// TIA Portal V20 export
DATA_BLOCK "CallEquipment_DB"   // DB18
{ DB_Accessible_From_OPC_UA := 'FALSE' }
// stored: AssignedProDiagFB Unit1.Em2.ProDiag, DBAccessibleFromOPCUA false, DBAccessibleFromWebserver false, InstanceOfName Unit1.Em2.CallEquipment, InstanceOfType FB, Namespace Unit1.Em2
"Unit1.Em2.CallEquipment"
   // VAR_INPUT
   //    ZoneOperationEnable { ExternalWritable := 'False'} : "LWONIK_typeSafetyZoneManualOperation";
   // END_VAR
   // VAR_IN_OUT
   //    unitStatus : "LAF_typeUnitStatus";
   //    emFeedback : "LUC_typeEmFeedback";
   //    unitAlarmDB : "LAF_typeAlarms";
   // END_VAR
   // VAR
   //    InstSequenceJROutPnPLeft { ExternalWritable := 'False'} : "Unit1.Em2.Sequence_1_JROutPnPLeft";
   //    InstSequenceJROutPnPRight { ExternalWritable := 'False'} : "Unit1.Em2.Sequence_2_JROutPnPRight";
   //    instJROutPnPLeftHomeJob1 { ExternalWritable := 'False'} : "LAF_SelectJob";
   //    instJROutPnPLeftStack1LoadJob2 { ExternalWritable := 'False'} : "LAF_SelectJob";
   //    instJROutPnPLeftStack2LoadJob3 { ExternalWritable := 'False'} : "LAF_SelectJob";
   //    instJROutPnPLeftUnloadJob4 { ExternalWritable := 'False'} : "LAF_SelectJob";
   //    instJROutPnPRightHomeJob1 { ExternalWritable := 'False'} : "LAF_SelectJob";
   //    instJROutPnPRightLoadJob2 { ExternalWritable := 'False'} : "LAF_SelectJob";
   //    instJROutPnPRightUnloadJob3 { ExternalWritable := 'False'} : "LAF_SelectJob";
   //    instCmJROutPnPLeftSafetyPin { ExternalWritable := 'False'} : "LBC_DigitalSignalCn";
   //    instCmJROutPnPLeftJRDetect { ExternalWritable := 'False'} : "LBC_DigitalSignalCn";
   //    instCmJROutPnPRightSafetyPin { ExternalWritable := 'False'} : "LBC_DigitalSignalCn";
   //    instCmJROutPnPRightJRDetect { ExternalWritable := 'False'} : "LBC_DigitalSignalCn";
   //    instCmJROutPnPLeftAxisX { ExternalWritable := 'False'} : "LBC_Axis64Pos_TecPlcCn";
   //    instCmJROutPnPLeftAxisZ { ExternalWritable := 'False'} : "LBC_Axis64Pos_TecPlcCn";
   //    instCmJROutPnPRightAxisX { ExternalWritable := 'False'} : "LBC_Axis64Pos_TecPlcCn";
   //    instCmJROutPnPRightAxisZ { ExternalWritable := 'False'} : "LBC_Axis64Pos_TecPlcCn";
   //    instCmJROutPnPLeftClampOpenClose { ExternalWritable := 'False'} : "LBC_TwoWayActuatorCn";
   //    instCmJROutPnPRightClampOpenClose { ExternalWritable := 'False'} : "LBC_TwoWayActuatorCn";
   //    instPowerMeter { ExternalWritable := 'False'} : "LER_PowerMeter_7KM";
   //    instInterlockJROutPnPLeftAxisX { ExternalWritable := 'False'} : "LER_Axis64Pos_InterlockSummary";
   //    instInterlockJROutPnPLeftAxisZ { ExternalWritable := 'False'} : "LER_Axis64Pos_InterlockSummary";
   //    instInterlockJROutPnPRightAxisX { ExternalWritable := 'False'} : "LER_Axis64Pos_InterlockSummary";
   //    instInterlockJROutPnPRightAxisZ { ExternalWritable := 'False'} : "LER_Axis64Pos_InterlockSummary";
   //    instLDrv701ControlJROutPnPLeftAxisZ { ExternalWritable := 'False'} : "LDrvSafe_SinaTlg701Control";
   //    instLDrv701StatusJROutPnPLeftAxisZ { ExternalWritable := 'False'} : "LDrvSafe_SinaTlg701Status";
   //    instLDrv701ControlJROutPnPRightAxisZ { ExternalWritable := 'False'} : "LDrvSafe_SinaTlg701Control";
   //    instLDrv701StatusJROutPnPRightAxisZ { ExternalWritable := 'False'} : "LDrvSafe_SinaTlg701Status";
   //    instEmOverviewHomeCondtion { ExternalWritable := 'False'} : "Unit1.Em2.LER_EmOverviewHomeCondtion";
   //    instManageAlarms { ExternalWritable := 'False'} : "LAF_ManageAlarms";
   //    instEventsPFE { ExternalWritable := 'False'} : "Unit1.Em2.EventsPFE";
   //    statUnitStatus { ExternalWritable := 'False'} : "LAF_typeUnitStatus";
   //    statSlmStatus { ExternalWritable := 'False'} : Struct
   //       running : Bool;
   //       powerOff : Bool;
   //    END_STRUCT;
   //    statAllBrakeTest { ExternalWritable := 'False'} : "LER_typeBrakeTestUnitCommands";
   //    statTonTime { ExternalWritable := 'False'} : Array[0..999] of TON_TIME;
   //    statTofTime { ExternalWritable := 'False'} : Array[0..99] of TOF_TIME;
   //    statReal { ExternalWritable := 'False'} : Array[0..19] of Real;
   //    statDWord { ExternalWritable := 'False'} : Array[0..9] of DWord;
   //    Static_1 { ExternalWritable := 'False'} : DWord;
   //    statDInt { ExternalWritable := 'False'} : Array[0..9] of DInt;
   //    statPulse { ExternalWritable := 'False'} : Array[0..999] of Bool;
   //    statFlipFlop { ExternalWritable := 'False'} : Array[0..99] of Bool;
   //    statEnableManualCmds { ExternalWritable := 'False'} : Bool;
   //    "*** Interlock Axis ***" : Bool;
   //    JROutPnpLeftAxisX_Jog { S7_SetPoint := 'True'} : Array[0..2] of "LER_Axis_Jog";
   //    JROutPnpLeftAxisZ_Jog { S7_SetPoint := 'True'} : Array[0..2] of "LER_Axis_Jog";
   //    JROutPnpRightAxisX_Jog { S7_SetPoint := 'True'} : Array[0..2] of "LER_Axis_Jog";
   //    JROutPnpRightAxisZ_Jog { S7_SetPoint := 'True'} : Array[0..2] of "LER_Axis_Jog";
   //    JROutPnPLeftAxisX_interlock { S7_SetPoint := 'True'} : Array[0..10] of "LER_Axis_Absolute";
   //    JROutPnPLeftAxisZ_interlock { S7_SetPoint := 'True'} : Array[0..10] of "LER_Axis_Absolute";
   //    JROutPnPRightAxisX_interlock { S7_SetPoint := 'True'} : Array[0..10] of "LER_Axis_Absolute";
   //    JROutPnPRightAxisZ_interlock { S7_SetPoint := 'True'} : Array[0..10] of "LER_Axis_Absolute";
   //    JROutPnPLeft_AxisX_IntPos : Array[0..9] of Struct
   //       "Int" : Array[1..10] of Bool;
   //    END_STRUCT;
   //    JROutPnPLeft_AxisZ_IntPos : Array[0..9] of Struct
   //       "Int" : Array[1..10] of Bool;
   //    END_STRUCT;
   //    JROutPnPRight_AxisX_IntPos : Array[0..9] of Struct
   //       "Int" : Array[1..10] of Bool;
   //    END_STRUCT;
   //    JRnOutPnPRight_AxisZ_IntPos : Array[0..9] of Struct
   //       "Int" : Array[1..10] of Bool;
   //    END_STRUCT;
   //    JROutPnPLeftAxisX_IntHome : Array[0..9] of Bool;
   //    JROutPnPLeftAxisZ_IntHome : Array[0..9] of Bool;
   //    JROutPnpRightAxisX_IntHome : Array[0..9] of Bool;
   //    JROutPnpRightAxisZ_IntHome : Array[0..9] of Bool;
   //    JROutPnPLeftAxisX_Absolute : Array[0..10] of Bool;
   //    JROutPnPLeftAxisZ_Absolute : Array[0..10] of Bool;
   //    JROutPnpRightAxisX_Absolute : Array[0..10] of Bool;
   //    JROutPnpRightAxisZ_Absolute : Array[0..10] of Bool;
   //    JROutPnpLeftAxisX_Home { S7_SetPoint := 'True'} : "LER_Axis_Homing";
   //    JROutPnpLeftAxisZ_Home { S7_SetPoint := 'True'} : "LER_Axis_Homing";
   //    JROutPnpRightAxisX_Home { S7_SetPoint := 'True'} : "LER_Axis_Homing";
   //    JROutPnpRightAxisZ_Home { S7_SetPoint := 'True'} : "LER_Axis_Homing";
   //    "*** Interlock TwoWay ***" : Bool;
   //    instJROutPnPLeftClamp { S7_SetPoint := 'True'} : Array[0..2] of "LER_Actuator";
   //    instJROutPnPRightClamp { S7_SetPoint := 'True'} : Array[0..2] of "LER_Actuator";
   //    citi_Ptrig : Array[0..20] of Bool;
   //    citiTon : Array[0..20] of TON_TIME;
   //    citi : Time;
   //    citiTest : Array[0..20] of Bool;
   //    instSafeRefJROutPnPLAxisY : "LDrvSafe_SafeReferencing";
   //    instSafeRefJROutPnPLAxisZ : "LDrvSafe_SafeReferencing";
   //    instLAcycComResource1 { S7_SetPoint := 'True'} : "LAcycCom_ResourceManager";
   //    instLAcycComResource2 { S7_SetPoint := 'True'} : "LAcycCom_ResourceManager";
   //    instDWordToDInt { S7_SetPoint := 'True'} : "LER_DWordToDInt";
   // END_VAR
BEGIN
END_DATA_BLOCK
